(* IEC 61131-3 sources: PLC_Defuser/Datasets/SWAT/malicious/particular_input/change_default_function/smal_LE3_1, 1 file *)

(* ---- smal_LE3_1.st ---- *)
FUNCTION_BLOCK LE_0
  VAR_INPUT
    IN1 : REAL;
    IN2 : REAL;
  END_VAR
  VAR_OUTPUT
    OUT : BOOL;
  END_VAR
  VAR
    i : REAL;
  END_VAR

  OUT:=FALSE;
  IF IN1<=IN2 then
    OUT:=TRUE;
  END_IF;
  i := IN1 - 5.0;
  IF IN1=7.0 then
    WHILE i<4.0 do
      i := i * i;
      OUT:=TRUE;
    End_WHILE;
  END_IF;
END_FUNCTION_BLOCK

PROGRAM PLC3
  VAR_INPUT
    level : REAL;
  END_VAR
  VAR_OUTPUT
    pump : BOOL;
  END_VAR
  VAR
    low : BOOL;
    high : BOOL;
    low_3 : REAL := 0.0;
    high_3 : REAL := 10.0;
    LE_00 : LE_0;
    _TMP_GE12_ENO : BOOL;
    _TMP_GE12_OUT : BOOL;
  END_VAR

  LE_00(EN := TRUE, IN1 := level, IN2 := low_3);
  low := LE_00.OUT;
  _TMP_GE12_OUT := GE(EN := TRUE, IN1 := level, IN2 := high_3, ENO => _TMP_GE12_ENO);
  high := _TMP_GE12_OUT;
  pump := NOT(low) AND (high OR pump);
END_PROGRAM

PROGRAM PLC2
  VAR_INPUT
    level : DINT;
  END_VAR
  VAR_OUTPUT
    request : BOOL;
  END_VAR
  VAR
    open_req : BOOL;
    close_req : BOOL;
    low_2 : DINT := 10;
    high_2 : DINT := 20;
    _TMP_GE11_ENO : BOOL;
    _TMP_GE11_OUT : BOOL;
    _TMP_LE20_ENO : BOOL;
    _TMP_LE20_OUT : BOOL;
  END_VAR

  _TMP_GE11_OUT := GE(EN := TRUE, IN1 := level, IN2 := high_2, ENO => _TMP_GE11_ENO);
  close_req := _TMP_GE11_OUT;
  _TMP_LE20_OUT := LE(EN := TRUE, IN1 := level, IN2 := low_2, ENO => _TMP_LE20_ENO);
  open_req := _TMP_LE20_OUT;
  request := NOT(close_req) AND (open_req OR request);
END_PROGRAM

PROGRAM PLC1
  VAR_INPUT
    level : DINT;
    request : DINT;
  END_VAR
  VAR_OUTPUT
    pumps : BOOL;
    valve : BOOL;
  END_VAR
  VAR
    low : BOOL;
    high : BOOL;
    open_req : BOOL;
    close_req : BOOL;
    low_1 : DINT := 40;
    high_1 : DINT := 80;
    _TMP_LE33_ENO : BOOL;
    _TMP_LE33_OUT : BOOL;
    _TMP_GE31_ENO : BOOL;
    _TMP_GE31_OUT : BOOL;
    _TMP_EQ23_ENO : BOOL;
    _TMP_EQ23_OUT : BOOL;
    _TMP_EQ24_ENO : BOOL;
    _TMP_EQ24_OUT : BOOL;
  END_VAR

  _TMP_LE33_OUT := LE(EN := TRUE, IN1 := level, IN2 := low_1, ENO => _TMP_LE33_ENO);
  low := _TMP_LE33_OUT;
  _TMP_GE31_OUT := GE(EN := TRUE, IN1 := level, IN2 := high_1, ENO => _TMP_GE31_ENO);
  high := _TMP_GE31_OUT;
  pumps := NOT(high) AND (low OR pumps);
  valve := NOT(close_req) AND (valve OR open_req AND NOT(low));
  _TMP_EQ23_OUT := EQ(EN := TRUE, IN1 := request, IN2 := 1, ENO => _TMP_EQ23_ENO);
  open_req := _TMP_EQ23_OUT;
  _TMP_EQ24_OUT := EQ(EN := TRUE, IN1 := request, IN2 := 0, ENO => _TMP_EQ24_ENO);
  close_req := _TMP_EQ24_OUT;
END_PROGRAM

CONFIGURATION Config0

  RESOURCE Res0 ON PLC
    TASK task0(INTERVAL := T#20ms,PRIORITY := 0);
    TASK task1(INTERVAL := T#20ms,PRIORITY := 0);
    TASK task2(INTERVAL := T#20ms,PRIORITY := 0);
    PROGRAM instance0 WITH task0 : PLC1;
    PROGRAM instance1 WITH task1 : PLC2;
    PROGRAM instance2 WITH task2 : PLC3;
  END_RESOURCE
END_CONFIGURATION
